PROGRAM START_STOP
VAR
	START_TIMER : TON;
	START_TIMER_ELAPSED: TIME;
	START_TIMER_DONE : BOOL; 
	ALARM_HORN AT %Q* : BOOL; // CONVEYOR STARTING WARNING SIGNAL
	ALL_CONVEYORS_START_PB  AT %I*:  BOOL; // TIE THIS TO THE START COMMAND FROM HMI OR BUTTON
	ALL_CONVEYORS_STOP_PB  AT %I*: BOOL; // TIE THIS TO THE STOP COMMAND FROM HMI OR BUTTON
	START_PB_LT AT %Q*: BOOL; // START PB LIGHT
	STOP_PB_LT AT %Q*: BOOL; // STOP PB LIGHT
	KIRK_BIT: BOOL;
	HMI_CONVEYOR_START: BOOL; // START SIGNAL FROM HMI
	
END_VAR

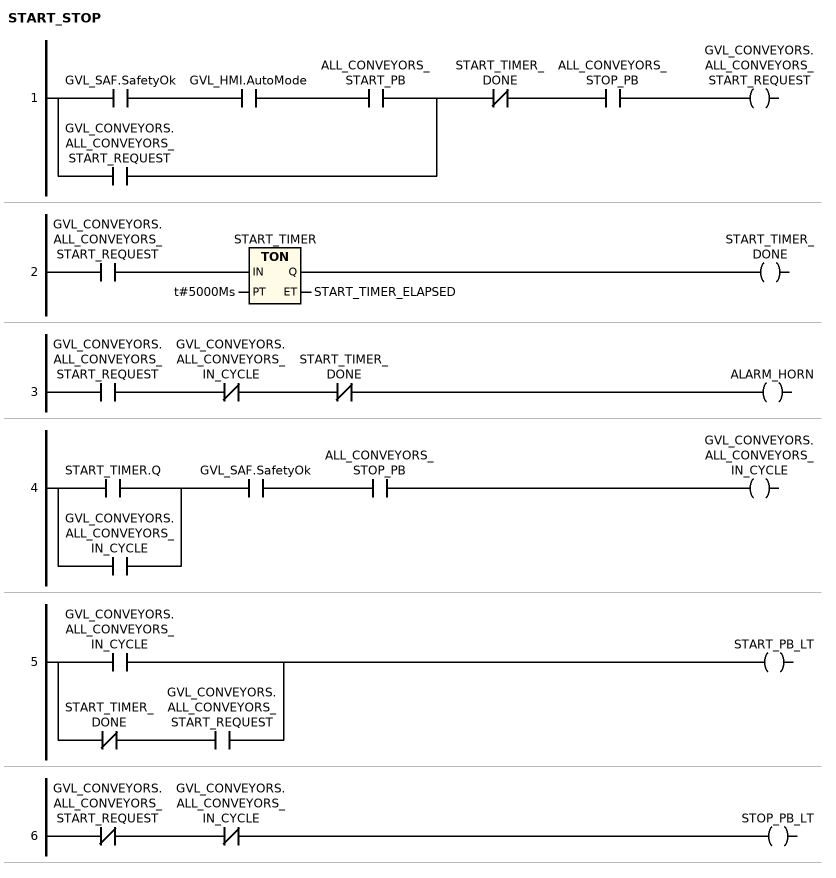
// NETWORK 1
GVL_CONVEYORS.ALL_CONVEYORS_START_REQUEST := (GVL_SAF.SafetyOk AND GVL_HMI.AutoMode AND ALL_CONVEYORS_START_PB OR GVL_CONVEYORS.ALL_CONVEYORS_START_REQUEST) AND NOT START_TIMER_DONE AND ALL_CONVEYORS_STOP_PB;

// NETWORK 2
START_TIMER(IN := GVL_CONVEYORS.ALL_CONVEYORS_START_REQUEST, PT := t#5000Ms, ET => START_TIMER_ELAPSED); // TON
START_TIMER_DONE := START_TIMER.Q;

// NETWORK 3
ALARM_HORN := GVL_CONVEYORS.ALL_CONVEYORS_START_REQUEST AND NOT GVL_CONVEYORS.ALL_CONVEYORS_IN_CYCLE AND NOT START_TIMER_DONE;

// NETWORK 4
GVL_CONVEYORS.ALL_CONVEYORS_IN_CYCLE := (START_TIMER.Q OR GVL_CONVEYORS.ALL_CONVEYORS_IN_CYCLE) AND GVL_SAF.SafetyOk AND ALL_CONVEYORS_STOP_PB;

// NETWORK 5
START_PB_LT := GVL_CONVEYORS.ALL_CONVEYORS_IN_CYCLE OR NOT START_TIMER_DONE AND GVL_CONVEYORS.ALL_CONVEYORS_START_REQUEST;

// NETWORK 6
STOP_PB_LT := NOT GVL_CONVEYORS.ALL_CONVEYORS_START_REQUEST AND NOT GVL_CONVEYORS.ALL_CONVEYORS_IN_CYCLE;

END_PROGRAM

(* stored: Version 1.1.0.1, ProductVersion 3.1.4024.12
   POU START_STOP: Id {0ade1615-2005-4f65-97b3-c1296d8b7762}, SpecialFunc None *)
